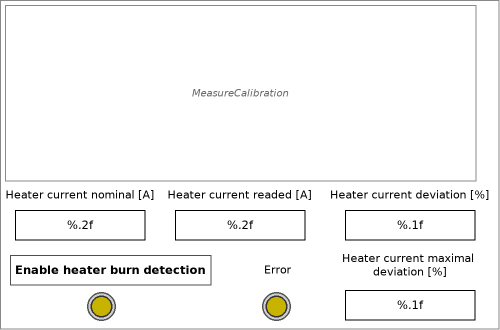
VISUALIZATION vHP3_WeldingPlateMonitorVisu  // 500x330
VAR_IN_OUT
	fbData	: fbHP_WeldPlateHeaterChecker;
END_VAR
    Rectangle (10,255 201x30), "Enable heater burn detection", colour toggle: fbData.stParams.bEnableWelderHeatersBurnDetection
        OnMouseClick: toggle fbData.stParams.bEnableWelderHeatersBurnDetection
    Rectangle (15,210 130x30), "%.2f", text variable: fbData.rCalculatedCurrentUsageValue
    Frame (5,5 471x176)
        shows MeasureCalibration(stMeasureData := fbData.stParams.stCalibrationData, diAnalogIn := fbData.iRawCurrentValue, MeasureName := 'Wedling Plate Current Scalling')
    Label (5,180 150x30), "Heater current nominal [A]"
    Label (165,180 150x30), "Heater current readed [A]"
    Label (325,180 170x30), "Heater current deviation [%]"
    Rectangle (175,210 130x30), "%.2f", text variable: fbData.rReadCurrentValue
    Rectangle (345,210 130x30), "%.1f", text variable: fbData.rDeviation
    Rectangle (345,290 130x30), "%.1f", text variable: fbData.stParams.rMaximalCurrentDeviation
        OnMouseClick: write the text variable via Default, min 5, max 100, format %1.f
    Label (335,240 150x50), "Heater current maximal deviation [%]"
    Lamp1 (85,290 33x33), variable: fbData.stParams.bEnableWelderHeatersBurnDetection, style: Lamp-Lamp1-Yellow
    Lamp1 (260,290 33x33), variable: fbData.bWeldingPlateHeaterError, style: Lamp-Lamp1-Yellow
    Label (235,255 85x30), "Error"
END_VISUALIZATION

(* stored: Version 1.1.0.1, ProductVersion 3.1.4024.15
   Visu vHP3_WeldingPlateMonitorVisu: Id {83296bd6-d9f2-4d8c-8a11-befed6565daa} *)
